{attribute 'strict'}
TYPE E_CSVDataExchangerCountColumnsState :
(
	CSV_DATA_EXCHANGER_COUNT_COLUMNS_OPEN_FILE 				:= 0,
	CSV_DATA_EXCHANGER_COUNT_COLUMNS_WAIT_FOR_OPENING		:= 10,	
	CSV_DATA_EXCHANGER_COUNT_COLUMNS_READ_SINGLE_LINE 		:= 20,	
	CSV_DATA_EXCHANGER_COUNT_COLUMNS_WAIT_FOR_READING		:= 30,	
	CSV_DATA_EXCHANGER_COUNT_COLUMNS_COUNT					:= 40,	
	CSV_DATA_EXCHANGER_COUNT_COLUMNS_CLOSE_FILE				:= 50,	
	CSV_DATA_EXCHANGER_COUNT_COLUMNS_WAIT_FOR_CLOSING		:= 60,
	CSV_DATA_EXCHANGER_COUNT_COLUMNS_READING_DONE			:= 70
);
END_TYPE

(* stored: Version 1.1.0.1, ProductVersion 3.1.4024.12
   DUT E_CSVDataExchangerCountColumnsState: Id {725e39f4-3141-4d75-b757-ef95e7b769ce} *)
